TYPE DUT_PARAMETER_INPUT :
STRUCT
	///Value of the parameter 
	Value: LREAL;
	///Possibility to a string value depending on the parameter
	StringValue: STRING(80);
END_STRUCT
END_TYPE

(* stored: Version 1.1.0.1, ProductVersion 3.1.0.25
   DUT DUT_PARAMETER_INPUT: Id {745e8eac-e7c1-4c70-8fbf-9ee97b2cd5ec} *)
